INTERFACE ITF_Observer

METHOD update : BOOL
VAR_INPUT
	Module : REFERENCE TO MachineModule;
END_VAR
END_METHOD

END_INTERFACE

(* stored: Version 1.1.0.1, ProductVersion 3.1.4024.12
   Itf ITF_Observer: Id {7fcd97c8-dddd-4c65-bfbc-c7a076a7a337}
   Method update: Id {c25919cf-b645-41c3-bb8f-6f088880249a} *)
